// TIA Portal V17 export
// export: Created 2025-04-09T08:02:46.8788876Z, ExportSetting WithDefaults, DisplayName Totally Integrated Automation Portal, DisplayVersion V17 Update 8, DisplayName TIA Portal Openness, DisplayVersion V17 Update 8, DisplayName TIA Portal Version Control Interface, DisplayVersion V17, DisplayName SINAMICS Startdrive Advanced, DisplayVersion V17 SP2, DisplayName SINAMICS Startdrive G110M, G120, G120C, G120D, G120P, G115D, DisplayVersion V17 SP2, DisplayName SINAMICS Startdrive G130, G150, S120, S150, SINAMICS MV, S210, DisplayVersion V17 SP2, DisplayName STEP 7 Professional, DisplayVersion V17 Update 8, DisplayName SINUMERIK ONE STEP 7 Toolbox, DisplayVersion V17 Update 12, DisplayName SINUMERIK ONE PLC Basic Program Plus, DisplayVersion V17 Update 12, DisplayName SINUMERIK 840D sl STEP 7 Toolbox, DisplayVersion V17 Update 12, DisplayName STEP 7 Safety, DisplayVersion V17 Update 6, DisplayName WinCC Advanced, DisplayVersion V17 Update 8
FUNCTION_BLOCK "FB1701_KELLER_ASPIRATION_CONTROL"   // FB1701, LAD
{ S7_Optimized_Access := 'TRUE' }
VERSION : 0.1
// stored: AutoNumber false, IsIECCheckEnabled false, IsRetainMemResEnabled false, MemoryReserve 100, SetENOAutomatically false, UDAEnableTagReadback false
   VAR_INPUT
      IN_PRODUCTION { ExternalAccessible := 'False'; ExternalVisible := 'False'; ExternalWritable := 'False'} : Bool;   // EXTRACTION IN PRODUCTION
      NOT_FAULT { ExternalAccessible := 'False'; ExternalVisible := 'False'; ExternalWritable := 'False'} : Bool;   // EXTRACTION OK
      REQ_FILTER_CLEAN { ExternalAccessible := 'False'; ExternalVisible := 'False'; ExternalWritable := 'False'} : Bool;   // REQUEST FILTER CLEAN
      HMI_REQ_LINE { ExternalAccessible := 'False'; ExternalVisible := 'False'; ExternalWritable := 'False'} : Bool;   // HMI REQUEST LINE
      MACHINE_ALARM : Bool;
   END_VAR
   VAR_OUTPUT
      SWITCH_ON { ExternalAccessible := 'False'; ExternalVisible := 'False'; ExternalWritable := 'False'} : Bool;   // EXTRACTION SWITCH ON
      MACHINE_OK { ExternalAccessible := 'False'; ExternalVisible := 'False'; ExternalWritable := 'False'} : Bool;   // MACHINE OK
      ALLOW_CLEANING { ExternalAccessible := 'False'; ExternalVisible := 'False'; ExternalWritable := 'False'} : Bool;   // EXTRACTION ALLOW CLEANING
      HMI_POWER_UP_COND_OFF : Bool;   // HMI POWER UP CONDITIONS OFF
      HMI_POWER_UP_COND_ON : Bool;   // HMI POWER UP CONDITIONS ON
      HMI_POWER_UP_EXECU_LEFT : Bool;   // HMI POWER UP EXECUTABLE LEFT
      HMI_POWER_UP_EXECU_RIGHT : Bool;   // HMI POWER UP EXECUTABLE RIGHT
   END_VAR
   VAR DB_SPECIFIC
      SWITCH_ON_GENERAL_CONDITIONS : Bool;   // SWITCH ON GENERAL CONDITIONS
      SWITCH_ON_INITIAL_CONDITIONS : Bool;   // SWITCH ON INITIAL CONDITIONS
      SWITCH_ON_MANUAL_REQUEST : Bool;   // SWITCH ON MANUAL REQUEST
      SWITCH_ON_AUTO_REQUEST : Bool;   // SWITCH ON AUTO REQUEST
      SWITCH_ON_GLOBAL_REQUEST : Bool;   // SWITCH ON GLOBAL REQUEST
      SWITCH_ON_COMMAND : Bool;   // SWITCH ON COMMAND
      SWITCH_ON_1 : Bool;   // SWITCH ON
      IN_SERVICE : Bool;   // IN SERVICE
      SWITCH_OFF_GENERAL_CONDITIONS : Bool;   // SWITCH OFF GENERAL CONDITIONS
      SWITCH_OFF_INITIAL_CONDITIONS : Bool;   // SWITCH OFF INITIAL CONDITIONS
      SWITCH_OFF_MANUAL_REQUEST : Bool;   // SWITCH OFF MANUAL REQUEST
      SWITCH_OFF_AUTO_REQUEST : Bool;   // SWITCH OFF AUTO REQUEST
      SWITCH_OFF_GLOBAL_REQUEST : Bool;   // SWITCH OFF GLOBAL REQUEST
      SWITCH_OFF_COMMAND : Bool;   // SWITCH OFF COMMAND
      SWITCH_OFF : Bool;   // SWITCH OFF
      OUT_OF_SERVICE : Bool;   // OUT OF SERVICE
      RUNOUT_REQ_CLEAN_FILTER : Bool;   // RUNOUT REQUEST BY ASPIRATION SYSTEM TO CLEAN FILTERS
      MANUAL_REQUEST_HELP : Bool;   // MANUAL REQUEST HELP
      SWITCH_ON_GENERAL_CONDITION_HELP : Bool;   // SWITCH ON GENERAL CONDITION HELP
      SWITCH_ON_INITIAL_CONDITION_HELP : Bool;   // SWITCH ON INITIAL CONDITION HELP
      SWITCH_OFF_GENERAL_CONDITION_HELP : Bool;   // SWITCH OFF GENERAL CONDITION HELP
      SWITCH_OFF_INITIAL_CONDITION_HELP : Bool;   // SWITCH OFF INITIAL CONDITION HELP
      EXTRACTION_ALARM : Bool;   // EXTRACTION IN FAULT STATE
      ANY_ACTIVE_ALARM : Bool;   // ANY ACTIVE ALARM
      IS_ALARMS : Bool;   // IMMEDIATE STOP ALARMS
      SEOC_ALARMS : Bool;   // STOP END OF CYCLE ALARMS
      WARNINGS : Bool;   // WARNINGS
      WARNINGS_GONE : Bool;   // WARNINGS GONE
   END_VAR
   VAR_TEMP
      DB_NUMBER : DInt;   // DB NUMBER FOR ALARM DECODING
   END_VAR
   VAR_TEMP   // added for the SCL form of the ladder/FBD networks
      _w1 : Bool;
   END_VAR
BEGIN

NETWORK
TITLE = READ INSTANCE DB
      L     DINO;
      +     10#800000;
      T     #DB_NUMBER;


REGION Network 2: SWITCH GENERAL CONDITIONS
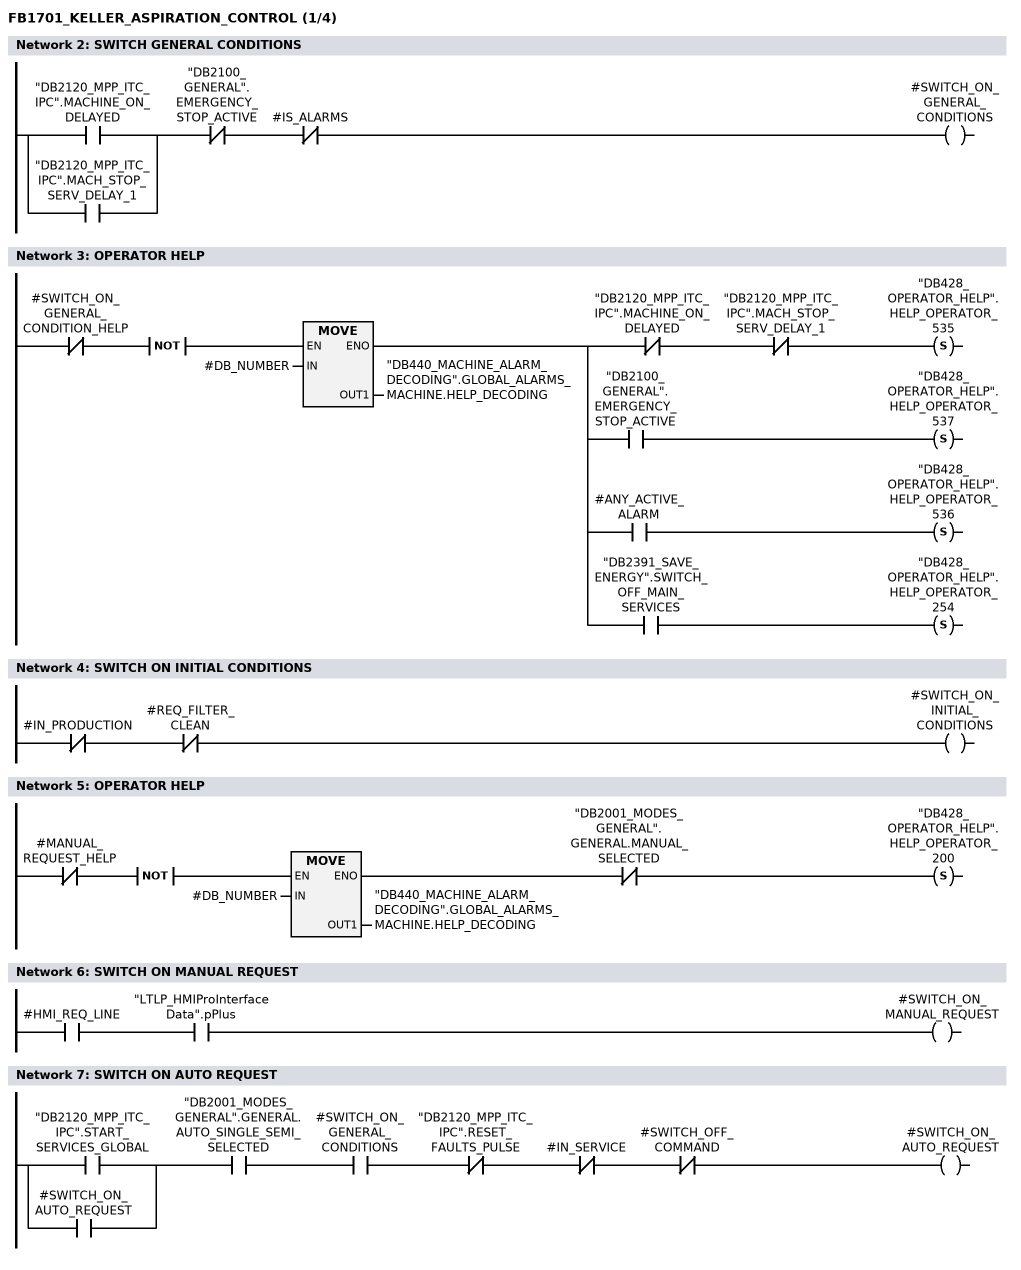
   RUNG wire#powerrail
      Contact( "DB2120_MPP_ITC_IPC".MACHINE_ON_DELAYED )
      wire#w1
      I_Contact( "DB2100_GENERAL".EMERGENCY_STOP_ACTIVE )
      I_Contact( #IS_ALARMS )
      Coil( #SWITCH_ON_GENERAL_CONDITIONS )
   END_RUNG
   RUNG wire#powerrail
      Contact( "DB2120_MPP_ITC_IPC".MACH_STOP_SERV_DELAY_1 )
   END_RUNG wire#w1
   // the same network as SCL:
   #SWITCH_ON_GENERAL_CONDITIONS := ("DB2120_MPP_ITC_IPC".MACHINE_ON_DELAYED OR "DB2120_MPP_ITC_IPC".MACH_STOP_SERV_DELAY_1) AND NOT "DB2100_GENERAL".EMERGENCY_STOP_ACTIVE AND NOT #IS_ALARMS;
END_REGION

REGION Network 3: OPERATOR HELP
   RUNG wire#powerrail
      I_Contact( #SWITCH_ON_GENERAL_CONDITION_HELP )
      Not()
      { S7_GenerateENO := "TRUE" } Move(in := #DB_NUMBER, out1 => "DB440_MACHINE_ALARM_DECODING".GLOBAL_ALARMS_MACHINE.HELP_DECODING)
      wire#w1
      I_Contact( "DB2120_MPP_ITC_IPC".MACHINE_ON_DELAYED )
      I_Contact( "DB2120_MPP_ITC_IPC".MACH_STOP_SERV_DELAY_1 )
      S_Coil( "DB428_OPERATOR_HELP".HELP_OPERATOR_535 )
   END_RUNG
   RUNG wire#w1
      Contact( "DB2100_GENERAL".EMERGENCY_STOP_ACTIVE )
      S_Coil( "DB428_OPERATOR_HELP".HELP_OPERATOR_537 )
   END_RUNG
   RUNG wire#w1
      Contact( #ANY_ACTIVE_ALARM )
      S_Coil( "DB428_OPERATOR_HELP".HELP_OPERATOR_536 )
   END_RUNG
   RUNG wire#w1
      Contact( "DB2391_SAVE_ENERGY".SWITCH_OFF_MAIN_SERVICES )
      S_Coil( "DB428_OPERATOR_HELP".HELP_OPERATOR_254 )
   END_RUNG
   // the same network as SCL:
   // ENO of a box is taken as its EN; it also drops when the box reports an error
   #_w1 := NOT (NOT #SWITCH_ON_GENERAL_CONDITION_HELP);
   IF #_w1 THEN "DB440_MACHINE_ALARM_DECODING".GLOBAL_ALARMS_MACHINE.HELP_DECODING := #DB_NUMBER; END_IF;
   IF #_w1 AND NOT "DB2120_MPP_ITC_IPC".MACHINE_ON_DELAYED AND NOT "DB2120_MPP_ITC_IPC".MACH_STOP_SERV_DELAY_1 THEN
       "DB428_OPERATOR_HELP".HELP_OPERATOR_535 := TRUE;
   END_IF;
   IF #_w1 AND "DB2100_GENERAL".EMERGENCY_STOP_ACTIVE THEN
       "DB428_OPERATOR_HELP".HELP_OPERATOR_537 := TRUE;
   END_IF;
   IF #_w1 AND #ANY_ACTIVE_ALARM THEN "DB428_OPERATOR_HELP".HELP_OPERATOR_536 := TRUE; END_IF;
   IF #_w1 AND "DB2391_SAVE_ENERGY".SWITCH_OFF_MAIN_SERVICES THEN
       "DB428_OPERATOR_HELP".HELP_OPERATOR_254 := TRUE;
   END_IF;
END_REGION

REGION Network 4: SWITCH ON INITIAL CONDITIONS
   RUNG wire#powerrail
      I_Contact( #IN_PRODUCTION )
      I_Contact( #REQ_FILTER_CLEAN )
      Coil( #SWITCH_ON_INITIAL_CONDITIONS )
   END_RUNG
   // the same network as SCL:
   #SWITCH_ON_INITIAL_CONDITIONS := NOT #IN_PRODUCTION AND NOT #REQ_FILTER_CLEAN;
END_REGION

REGION Network 5: OPERATOR HELP
   RUNG wire#powerrail
      I_Contact( #MANUAL_REQUEST_HELP )
      Not()
      { S7_GenerateENO := "TRUE" } Move(in := #DB_NUMBER, out1 => "DB440_MACHINE_ALARM_DECODING".GLOBAL_ALARMS_MACHINE.HELP_DECODING)
      I_Contact( "DB2001_MODES_GENERAL".GENERAL.MANUAL_SELECTED )
      S_Coil( "DB428_OPERATOR_HELP".HELP_OPERATOR_200 )
   END_RUNG
   // the same network as SCL:
   // ENO of a box is taken as its EN; it also drops when the box reports an error
   #_w1 := NOT (NOT #MANUAL_REQUEST_HELP);
   IF #_w1 THEN "DB440_MACHINE_ALARM_DECODING".GLOBAL_ALARMS_MACHINE.HELP_DECODING := #DB_NUMBER; END_IF;
   IF #_w1 AND NOT "DB2001_MODES_GENERAL".GENERAL.MANUAL_SELECTED THEN
       "DB428_OPERATOR_HELP".HELP_OPERATOR_200 := TRUE;
   END_IF;
END_REGION

REGION Network 6: SWITCH ON MANUAL REQUEST
   RUNG wire#powerrail
      Contact( #HMI_REQ_LINE )
      Contact( "LTLP_HMIProInterfaceData".pPlus )
      Coil( #SWITCH_ON_MANUAL_REQUEST )
   END_RUNG
   // the same network as SCL:
   #SWITCH_ON_MANUAL_REQUEST := #HMI_REQ_LINE AND "LTLP_HMIProInterfaceData".pPlus;
END_REGION

REGION Network 7: SWITCH ON AUTO REQUEST
   RUNG wire#powerrail
      Contact( "DB2120_MPP_ITC_IPC".START_SERVICES_GLOBAL )
      wire#w1
      Contact( "DB2001_MODES_GENERAL".GENERAL.AUTO_SINGLE_SEMI_SELECTED )
      Contact( #SWITCH_ON_GENERAL_CONDITIONS )
      I_Contact( "DB2120_MPP_ITC_IPC".RESET_FAULTS_PULSE )
      I_Contact( #IN_SERVICE )
      I_Contact( #SWITCH_OFF_COMMAND )
      Coil( #SWITCH_ON_AUTO_REQUEST )
   END_RUNG
   RUNG wire#powerrail
      Contact( #SWITCH_ON_AUTO_REQUEST )
   END_RUNG wire#w1
   // the same network as SCL:
   #SWITCH_ON_AUTO_REQUEST := ("DB2120_MPP_ITC_IPC".START_SERVICES_GLOBAL OR #SWITCH_ON_AUTO_REQUEST) AND "DB2001_MODES_GENERAL".GENERAL.AUTO_SINGLE_SEMI_SELECTED AND #SWITCH_ON_GENERAL_CONDITIONS AND NOT "DB2120_MPP_ITC_IPC".RESET_FAULTS_PULSE AND NOT #IN_SERVICE AND NOT #SWITCH_OFF_COMMAND;
END_REGION

REGION Network 8: SWITCH ON GLOBAL REQUEST
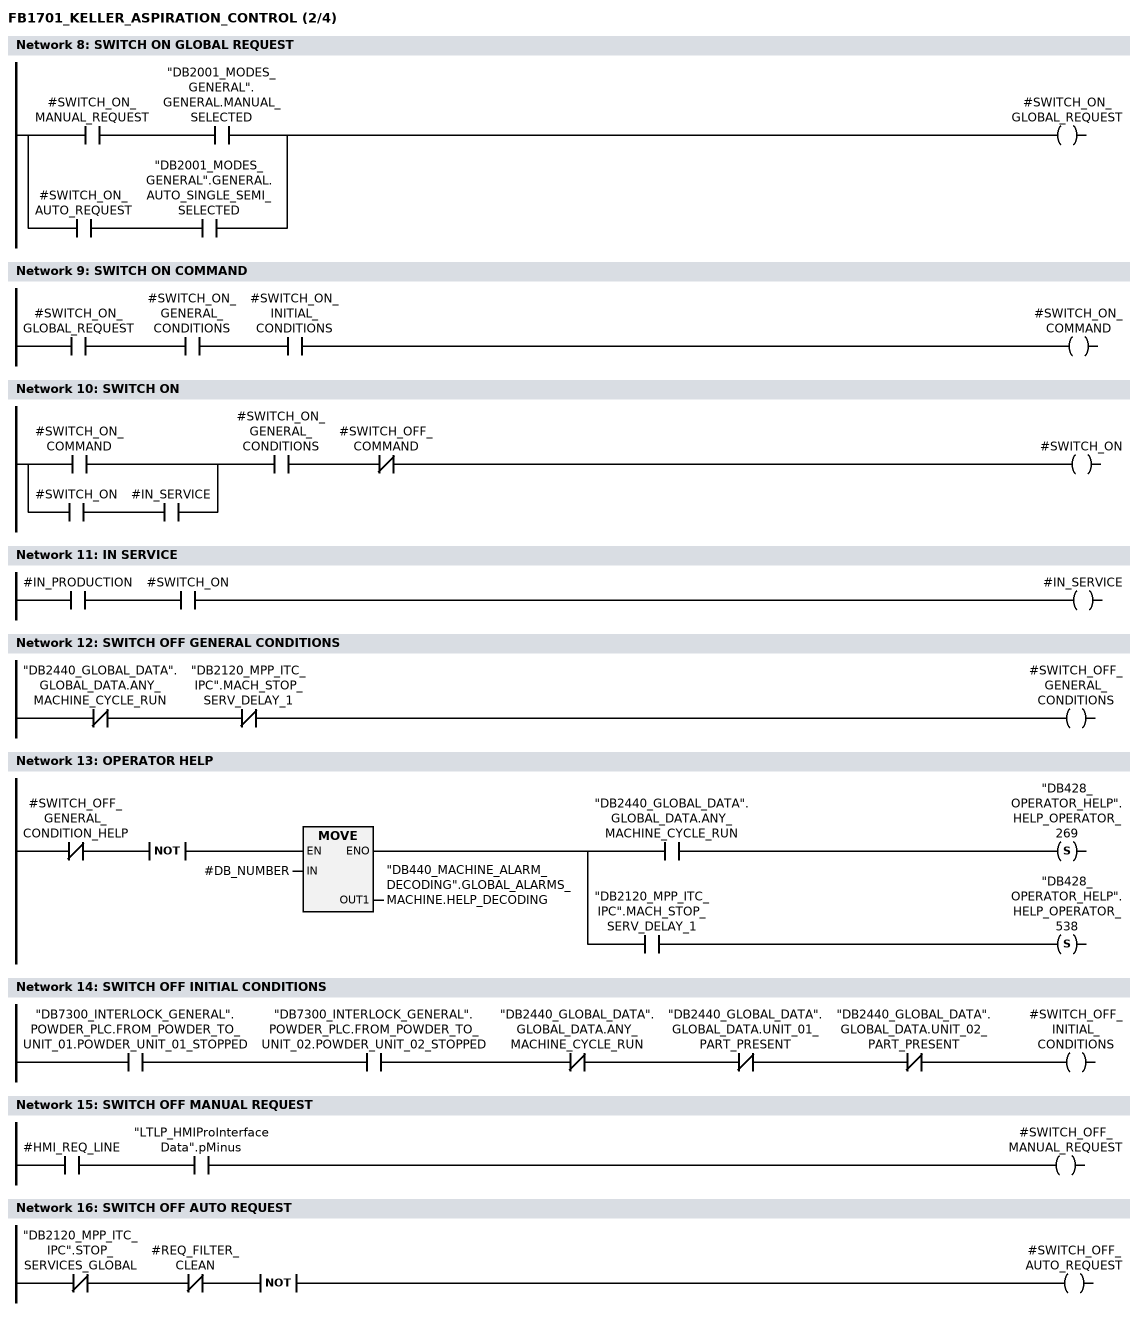
   RUNG wire#powerrail
      Contact( #SWITCH_ON_MANUAL_REQUEST )
      Contact( "DB2001_MODES_GENERAL".GENERAL.MANUAL_SELECTED )
      wire#w1
      Coil( #SWITCH_ON_GLOBAL_REQUEST )
   END_RUNG
   RUNG wire#powerrail
      Contact( #SWITCH_ON_AUTO_REQUEST )
      Contact( "DB2001_MODES_GENERAL".GENERAL.AUTO_SINGLE_SEMI_SELECTED )
   END_RUNG wire#w1
   // the same network as SCL:
   #SWITCH_ON_GLOBAL_REQUEST := (#SWITCH_ON_MANUAL_REQUEST AND "DB2001_MODES_GENERAL".GENERAL.MANUAL_SELECTED) OR (#SWITCH_ON_AUTO_REQUEST AND "DB2001_MODES_GENERAL".GENERAL.AUTO_SINGLE_SEMI_SELECTED);
END_REGION

REGION Network 9: SWITCH ON COMMAND
   RUNG wire#powerrail
      Contact( #SWITCH_ON_GLOBAL_REQUEST )
      Contact( #SWITCH_ON_GENERAL_CONDITIONS )
      Contact( #SWITCH_ON_INITIAL_CONDITIONS )
      Coil( #SWITCH_ON_COMMAND )
   END_RUNG
   // the same network as SCL:
   #SWITCH_ON_COMMAND := #SWITCH_ON_GLOBAL_REQUEST AND #SWITCH_ON_GENERAL_CONDITIONS AND #SWITCH_ON_INITIAL_CONDITIONS;
END_REGION

REGION Network 10: SWITCH ON
   RUNG wire#powerrail
      Contact( #SWITCH_ON_COMMAND )
      wire#w1
      Contact( #SWITCH_ON_GENERAL_CONDITIONS )
      I_Contact( #SWITCH_OFF_COMMAND )
      Coil( #SWITCH_ON )
   END_RUNG
   RUNG wire#powerrail
      Contact( #SWITCH_ON )
      Contact( #IN_SERVICE )
   END_RUNG wire#w1
   // the same network as SCL:
   #SWITCH_ON := (#SWITCH_ON_COMMAND OR (#SWITCH_ON AND #IN_SERVICE)) AND #SWITCH_ON_GENERAL_CONDITIONS AND NOT #SWITCH_OFF_COMMAND;
END_REGION

REGION Network 11: IN SERVICE
   RUNG wire#powerrail
      Contact( #IN_PRODUCTION )
      Contact( #SWITCH_ON )
      Coil( #IN_SERVICE )
   END_RUNG
   // the same network as SCL:
   #IN_SERVICE := #IN_PRODUCTION AND #SWITCH_ON;
END_REGION

REGION Network 12: SWITCH OFF GENERAL CONDITIONS
   RUNG wire#powerrail
      I_Contact( "DB2440_GLOBAL_DATA".GLOBAL_DATA.ANY_MACHINE_CYCLE_RUN )
      I_Contact( "DB2120_MPP_ITC_IPC".MACH_STOP_SERV_DELAY_1 )
      Coil( #SWITCH_OFF_GENERAL_CONDITIONS )
   END_RUNG
   // the same network as SCL:
   #SWITCH_OFF_GENERAL_CONDITIONS := NOT "DB2440_GLOBAL_DATA".GLOBAL_DATA.ANY_MACHINE_CYCLE_RUN AND NOT "DB2120_MPP_ITC_IPC".MACH_STOP_SERV_DELAY_1;
END_REGION

REGION Network 13: OPERATOR HELP
   RUNG wire#powerrail
      I_Contact( #SWITCH_OFF_GENERAL_CONDITION_HELP )
      Not()
      { S7_GenerateENO := "TRUE" } Move(in := #DB_NUMBER, out1 => "DB440_MACHINE_ALARM_DECODING".GLOBAL_ALARMS_MACHINE.HELP_DECODING)
      wire#w1
      Contact( "DB2440_GLOBAL_DATA".GLOBAL_DATA.ANY_MACHINE_CYCLE_RUN )
      S_Coil( "DB428_OPERATOR_HELP".HELP_OPERATOR_269 )
   END_RUNG
   RUNG wire#w1
      Contact( "DB2120_MPP_ITC_IPC".MACH_STOP_SERV_DELAY_1 )
      S_Coil( "DB428_OPERATOR_HELP".HELP_OPERATOR_538 )
   END_RUNG
   // the same network as SCL:
   // ENO of a box is taken as its EN; it also drops when the box reports an error
   #_w1 := NOT (NOT #SWITCH_OFF_GENERAL_CONDITION_HELP);
   IF #_w1 THEN "DB440_MACHINE_ALARM_DECODING".GLOBAL_ALARMS_MACHINE.HELP_DECODING := #DB_NUMBER; END_IF;
   IF #_w1 AND "DB2440_GLOBAL_DATA".GLOBAL_DATA.ANY_MACHINE_CYCLE_RUN THEN
       "DB428_OPERATOR_HELP".HELP_OPERATOR_269 := TRUE;
   END_IF;
   IF #_w1 AND "DB2120_MPP_ITC_IPC".MACH_STOP_SERV_DELAY_1 THEN
       "DB428_OPERATOR_HELP".HELP_OPERATOR_538 := TRUE;
   END_IF;
END_REGION

REGION Network 14: SWITCH OFF INITIAL CONDITIONS
   RUNG wire#powerrail
      Contact( "DB7300_INTERLOCK_GENERAL".POWDER_PLC.FROM_POWDER_TO_UNIT_01.POWDER_UNIT_01_STOPPED )
      Contact( "DB7300_INTERLOCK_GENERAL".POWDER_PLC.FROM_POWDER_TO_UNIT_02.POWDER_UNIT_02_STOPPED )
      I_Contact( "DB2440_GLOBAL_DATA".GLOBAL_DATA.ANY_MACHINE_CYCLE_RUN )
      I_Contact( "DB2440_GLOBAL_DATA".GLOBAL_DATA.UNIT_01_PART_PRESENT )
      I_Contact( "DB2440_GLOBAL_DATA".GLOBAL_DATA.UNIT_02_PART_PRESENT )
      Coil( #SWITCH_OFF_INITIAL_CONDITIONS )
   END_RUNG
   // the same network as SCL:
   #SWITCH_OFF_INITIAL_CONDITIONS := "DB7300_INTERLOCK_GENERAL".POWDER_PLC.FROM_POWDER_TO_UNIT_01.POWDER_UNIT_01_STOPPED AND "DB7300_INTERLOCK_GENERAL".POWDER_PLC.FROM_POWDER_TO_UNIT_02.POWDER_UNIT_02_STOPPED AND NOT "DB2440_GLOBAL_DATA".GLOBAL_DATA.ANY_MACHINE_CYCLE_RUN AND NOT "DB2440_GLOBAL_DATA".GLOBAL_DATA.UNIT_01_PART_PRESENT AND NOT "DB2440_GLOBAL_DATA".GLOBAL_DATA.UNIT_02_PART_PRESENT;
END_REGION

REGION Network 15: SWITCH OFF MANUAL REQUEST
   RUNG wire#powerrail
      Contact( #HMI_REQ_LINE )
      Contact( "LTLP_HMIProInterfaceData".pMinus )
      Coil( #SWITCH_OFF_MANUAL_REQUEST )
   END_RUNG
   // the same network as SCL:
   #SWITCH_OFF_MANUAL_REQUEST := #HMI_REQ_LINE AND "LTLP_HMIProInterfaceData".pMinus;
END_REGION

REGION Network 16: SWITCH OFF AUTO REQUEST
   RUNG wire#powerrail
      I_Contact( "DB2120_MPP_ITC_IPC".STOP_SERVICES_GLOBAL )
      I_Contact( #REQ_FILTER_CLEAN )
      Not()
      Coil( #SWITCH_OFF_AUTO_REQUEST )
   END_RUNG
   // the same network as SCL:
   #SWITCH_OFF_AUTO_REQUEST := NOT (NOT "DB2120_MPP_ITC_IPC".STOP_SERVICES_GLOBAL AND NOT #REQ_FILTER_CLEAN);
END_REGION

REGION Network 17: SWITCH OFF GLOBAL REQUEST
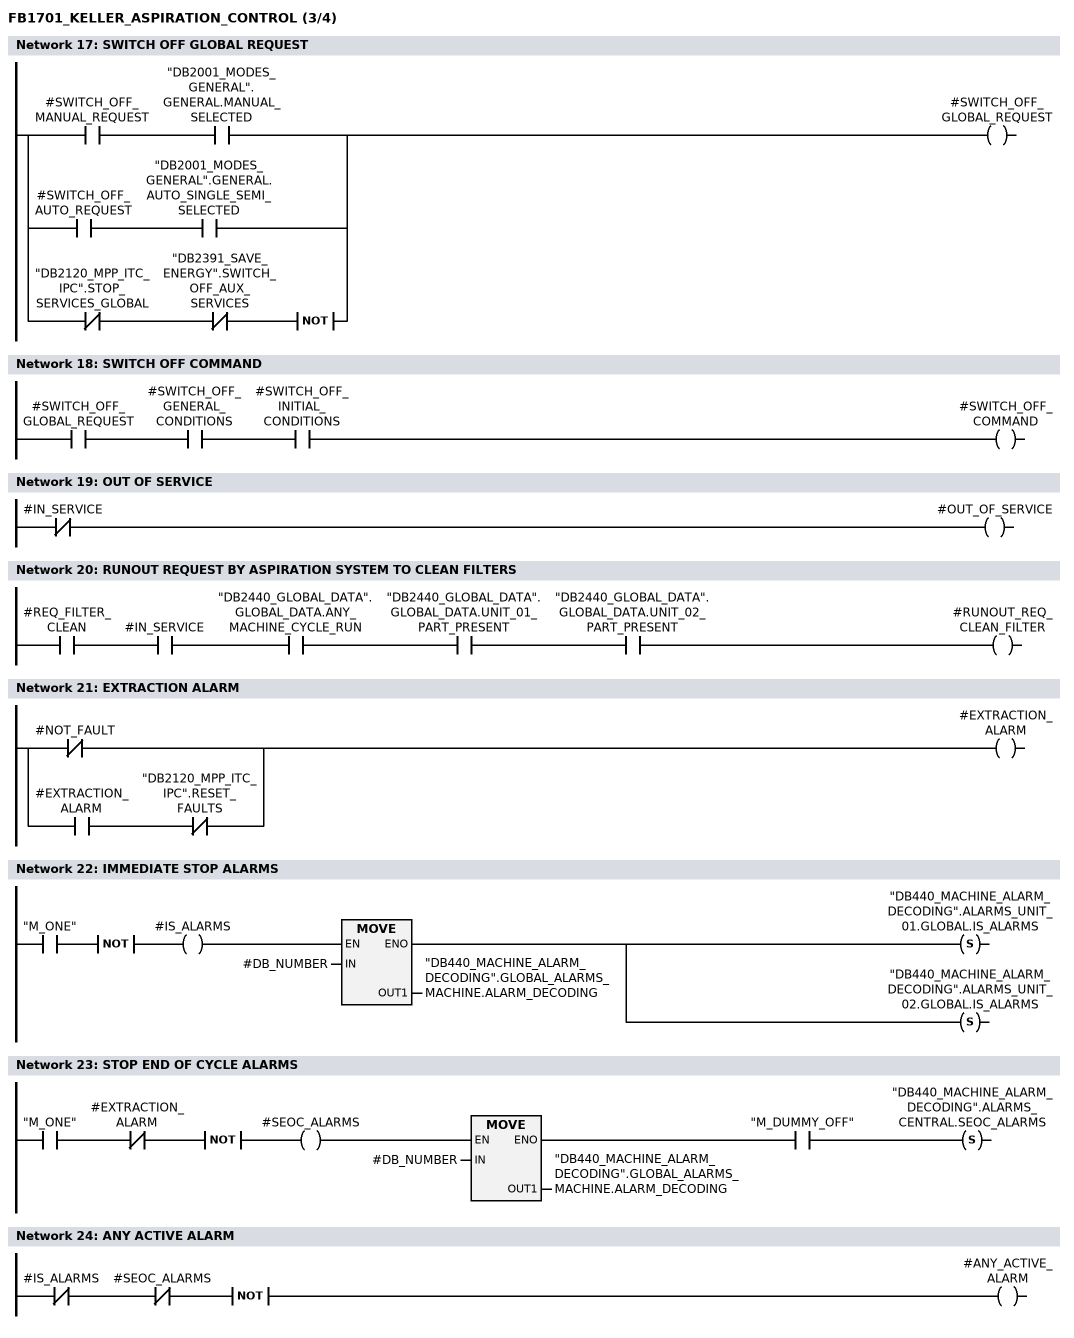
   RUNG wire#powerrail
      Contact( #SWITCH_OFF_MANUAL_REQUEST )
      Contact( "DB2001_MODES_GENERAL".GENERAL.MANUAL_SELECTED )
      wire#w1
      Coil( #SWITCH_OFF_GLOBAL_REQUEST )
   END_RUNG
   RUNG wire#powerrail
      Contact( #SWITCH_OFF_AUTO_REQUEST )
      Contact( "DB2001_MODES_GENERAL".GENERAL.AUTO_SINGLE_SEMI_SELECTED )
   END_RUNG wire#w1
   RUNG wire#powerrail
      I_Contact( "DB2120_MPP_ITC_IPC".STOP_SERVICES_GLOBAL )
      I_Contact( "DB2391_SAVE_ENERGY".SWITCH_OFF_AUX_SERVICES )
      Not()
   END_RUNG wire#w1
   // the same network as SCL:
   #SWITCH_OFF_GLOBAL_REQUEST := (#SWITCH_OFF_MANUAL_REQUEST AND "DB2001_MODES_GENERAL".GENERAL.MANUAL_SELECTED) OR (#SWITCH_OFF_AUTO_REQUEST AND "DB2001_MODES_GENERAL".GENERAL.AUTO_SINGLE_SEMI_SELECTED) OR NOT (NOT "DB2120_MPP_ITC_IPC".STOP_SERVICES_GLOBAL AND NOT "DB2391_SAVE_ENERGY".SWITCH_OFF_AUX_SERVICES);
END_REGION

REGION Network 18: SWITCH OFF COMMAND
   RUNG wire#powerrail
      Contact( #SWITCH_OFF_GLOBAL_REQUEST )
      Contact( #SWITCH_OFF_GENERAL_CONDITIONS )
      Contact( #SWITCH_OFF_INITIAL_CONDITIONS )
      Coil( #SWITCH_OFF_COMMAND )
   END_RUNG
   // the same network as SCL:
   #SWITCH_OFF_COMMAND := #SWITCH_OFF_GLOBAL_REQUEST AND #SWITCH_OFF_GENERAL_CONDITIONS AND #SWITCH_OFF_INITIAL_CONDITIONS;
END_REGION

REGION Network 19: OUT OF SERVICE
   RUNG wire#powerrail
      I_Contact( #IN_SERVICE )
      Coil( #OUT_OF_SERVICE )
   END_RUNG
   // the same network as SCL:
   #OUT_OF_SERVICE := NOT #IN_SERVICE;
END_REGION

REGION Network 20: RUNOUT REQUEST BY ASPIRATION SYSTEM TO CLEAN FILTERS
   RUNG wire#powerrail
      Contact( #REQ_FILTER_CLEAN )
      Contact( #IN_SERVICE )
      Contact( "DB2440_GLOBAL_DATA".GLOBAL_DATA.ANY_MACHINE_CYCLE_RUN )
      Contact( "DB2440_GLOBAL_DATA".GLOBAL_DATA.UNIT_01_PART_PRESENT )
      Contact( "DB2440_GLOBAL_DATA".GLOBAL_DATA.UNIT_02_PART_PRESENT )
      Coil( #RUNOUT_REQ_CLEAN_FILTER )
   END_RUNG
   // the same network as SCL:
   #RUNOUT_REQ_CLEAN_FILTER := #REQ_FILTER_CLEAN AND #IN_SERVICE AND "DB2440_GLOBAL_DATA".GLOBAL_DATA.ANY_MACHINE_CYCLE_RUN AND "DB2440_GLOBAL_DATA".GLOBAL_DATA.UNIT_01_PART_PRESENT AND "DB2440_GLOBAL_DATA".GLOBAL_DATA.UNIT_02_PART_PRESENT;
END_REGION

REGION Network 21: EXTRACTION ALARM
   RUNG wire#powerrail
      I_Contact( #NOT_FAULT )
      wire#w1
      Coil( #EXTRACTION_ALARM )
   END_RUNG
   RUNG wire#powerrail
      Contact( #EXTRACTION_ALARM )
      I_Contact( "DB2120_MPP_ITC_IPC".RESET_FAULTS )
   END_RUNG wire#w1
   // the same network as SCL:
   #EXTRACTION_ALARM := NOT #NOT_FAULT OR (#EXTRACTION_ALARM AND NOT "DB2120_MPP_ITC_IPC".RESET_FAULTS);
END_REGION

REGION Network 22: IMMEDIATE STOP ALARMS
   RUNG wire#powerrail
      Contact( "M_ONE" )
      Not()
      Coil( #IS_ALARMS )
      Move(in := #DB_NUMBER, out1 => "DB440_MACHINE_ALARM_DECODING".GLOBAL_ALARMS_MACHINE.ALARM_DECODING)
      wire#w1
      S_Coil( "DB440_MACHINE_ALARM_DECODING".ALARMS_UNIT_01.GLOBAL.IS_ALARMS )
   END_RUNG
   RUNG wire#w1
      S_Coil( "DB440_MACHINE_ALARM_DECODING".ALARMS_UNIT_02.GLOBAL.IS_ALARMS )
   END_RUNG
   // the same network as SCL:
   #IS_ALARMS := NOT "M_ONE";
   IF NOT "M_ONE" THEN
       "DB440_MACHINE_ALARM_DECODING".GLOBAL_ALARMS_MACHINE.ALARM_DECODING := #DB_NUMBER;
       "DB440_MACHINE_ALARM_DECODING".ALARMS_UNIT_01.GLOBAL.IS_ALARMS := TRUE;
       "DB440_MACHINE_ALARM_DECODING".ALARMS_UNIT_02.GLOBAL.IS_ALARMS := TRUE;
   END_IF;
END_REGION

REGION Network 23: STOP END OF CYCLE ALARMS
   RUNG wire#powerrail
      Contact( "M_ONE" )
      I_Contact( #EXTRACTION_ALARM )
      Not()
      Coil( #SEOC_ALARMS )
      Move(in := #DB_NUMBER, out1 => "DB440_MACHINE_ALARM_DECODING".GLOBAL_ALARMS_MACHINE.ALARM_DECODING)
      Contact( "M_DUMMY_OFF" )
      S_Coil( "DB440_MACHINE_ALARM_DECODING".ALARMS_CENTRAL.SEOC_ALARMS )
   END_RUNG
   // the same network as SCL:
   #SEOC_ALARMS := NOT ("M_ONE" AND NOT #EXTRACTION_ALARM);
   IF #SEOC_ALARMS THEN
       "DB440_MACHINE_ALARM_DECODING".GLOBAL_ALARMS_MACHINE.ALARM_DECODING := #DB_NUMBER;
   END_IF;
   IF #SEOC_ALARMS AND "M_DUMMY_OFF" THEN
       "DB440_MACHINE_ALARM_DECODING".ALARMS_CENTRAL.SEOC_ALARMS := TRUE;
   END_IF;
END_REGION

REGION Network 24: ANY ACTIVE ALARM
   RUNG wire#powerrail
      I_Contact( #IS_ALARMS )
      I_Contact( #SEOC_ALARMS )
      Not()
      Coil( #ANY_ACTIVE_ALARM )
   END_RUNG
   // the same network as SCL:
   #ANY_ACTIVE_ALARM := NOT (NOT #IS_ALARMS AND NOT #SEOC_ALARMS);
END_REGION

REGION Network 25: MANUAL REQUEST HELP
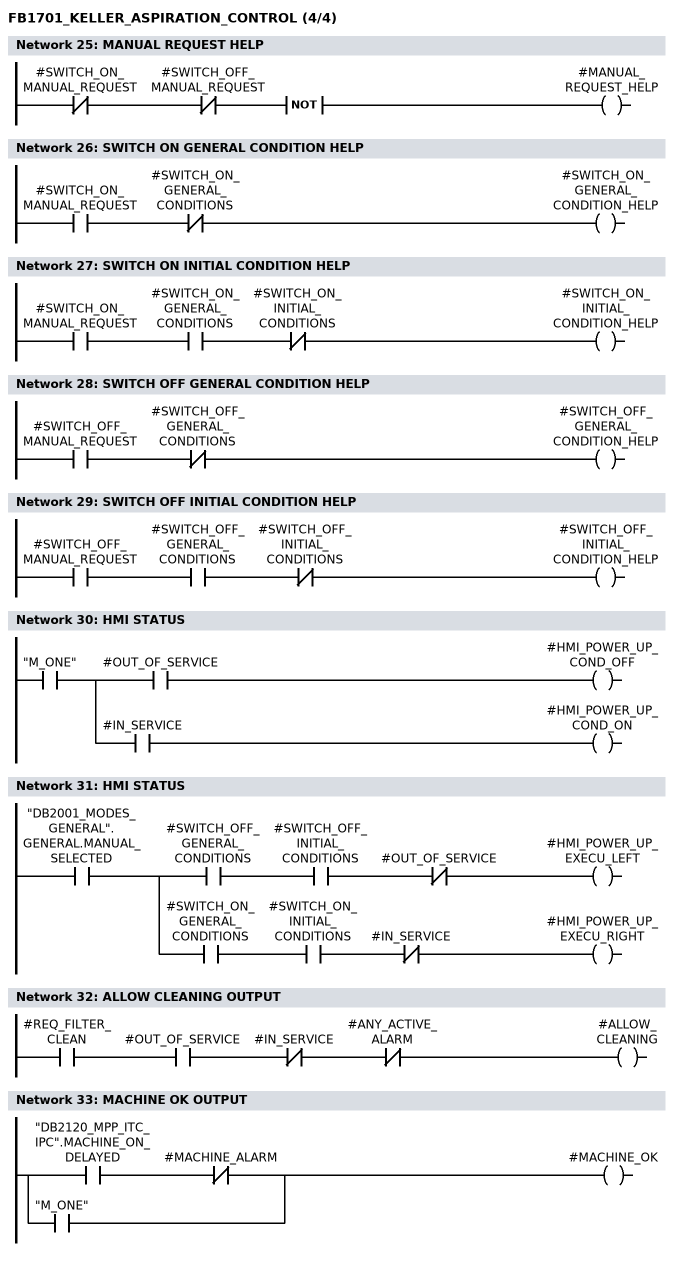
   RUNG wire#powerrail
      I_Contact( #SWITCH_ON_MANUAL_REQUEST )
      I_Contact( #SWITCH_OFF_MANUAL_REQUEST )
      Not()
      Coil( #MANUAL_REQUEST_HELP )
   END_RUNG
   // the same network as SCL:
   #MANUAL_REQUEST_HELP := NOT (NOT #SWITCH_ON_MANUAL_REQUEST AND NOT #SWITCH_OFF_MANUAL_REQUEST);
END_REGION

REGION Network 26: SWITCH ON GENERAL CONDITION HELP
   RUNG wire#powerrail
      Contact( #SWITCH_ON_MANUAL_REQUEST )
      I_Contact( #SWITCH_ON_GENERAL_CONDITIONS )
      Coil( #SWITCH_ON_GENERAL_CONDITION_HELP )
   END_RUNG
   // the same network as SCL:
   #SWITCH_ON_GENERAL_CONDITION_HELP := #SWITCH_ON_MANUAL_REQUEST AND NOT #SWITCH_ON_GENERAL_CONDITIONS;
END_REGION

REGION Network 27: SWITCH ON INITIAL CONDITION HELP
   RUNG wire#powerrail
      Contact( #SWITCH_ON_MANUAL_REQUEST )
      Contact( #SWITCH_ON_GENERAL_CONDITIONS )
      I_Contact( #SWITCH_ON_INITIAL_CONDITIONS )
      Coil( #SWITCH_ON_INITIAL_CONDITION_HELP )
   END_RUNG
   // the same network as SCL:
   #SWITCH_ON_INITIAL_CONDITION_HELP := #SWITCH_ON_MANUAL_REQUEST AND #SWITCH_ON_GENERAL_CONDITIONS AND NOT #SWITCH_ON_INITIAL_CONDITIONS;
END_REGION

REGION Network 28: SWITCH OFF GENERAL CONDITION HELP
   RUNG wire#powerrail
      Contact( #SWITCH_OFF_MANUAL_REQUEST )
      I_Contact( #SWITCH_OFF_GENERAL_CONDITIONS )
      Coil( #SWITCH_OFF_GENERAL_CONDITION_HELP )
   END_RUNG
   // the same network as SCL:
   #SWITCH_OFF_GENERAL_CONDITION_HELP := #SWITCH_OFF_MANUAL_REQUEST AND NOT #SWITCH_OFF_GENERAL_CONDITIONS;
END_REGION

REGION Network 29: SWITCH OFF INITIAL CONDITION HELP
   RUNG wire#powerrail
      Contact( #SWITCH_OFF_MANUAL_REQUEST )
      Contact( #SWITCH_OFF_GENERAL_CONDITIONS )
      I_Contact( #SWITCH_OFF_INITIAL_CONDITIONS )
      Coil( #SWITCH_OFF_INITIAL_CONDITION_HELP )
   END_RUNG
   // the same network as SCL:
   #SWITCH_OFF_INITIAL_CONDITION_HELP := #SWITCH_OFF_MANUAL_REQUEST AND #SWITCH_OFF_GENERAL_CONDITIONS AND NOT #SWITCH_OFF_INITIAL_CONDITIONS;
END_REGION

REGION Network 30: HMI STATUS
   RUNG wire#powerrail
      Contact( "M_ONE" )
      wire#w1
      Contact( #OUT_OF_SERVICE )
      Coil( #HMI_POWER_UP_COND_OFF )
   END_RUNG
   RUNG wire#w1
      Contact( #IN_SERVICE )
      Coil( #HMI_POWER_UP_COND_ON )
   END_RUNG
   // the same network as SCL:
   #HMI_POWER_UP_COND_OFF := "M_ONE" AND #OUT_OF_SERVICE;
   #HMI_POWER_UP_COND_ON := "M_ONE" AND #IN_SERVICE;
END_REGION

REGION Network 31: HMI STATUS
   RUNG wire#powerrail
      Contact( "DB2001_MODES_GENERAL".GENERAL.MANUAL_SELECTED )
      wire#w1
      Contact( #SWITCH_OFF_GENERAL_CONDITIONS )
      Contact( #SWITCH_OFF_INITIAL_CONDITIONS )
      I_Contact( #OUT_OF_SERVICE )
      Coil( #HMI_POWER_UP_EXECU_LEFT )
   END_RUNG
   RUNG wire#w1
      Contact( #SWITCH_ON_GENERAL_CONDITIONS )
      Contact( #SWITCH_ON_INITIAL_CONDITIONS )
      I_Contact( #IN_SERVICE )
      Coil( #HMI_POWER_UP_EXECU_RIGHT )
   END_RUNG
   // the same network as SCL:
   #HMI_POWER_UP_EXECU_LEFT := "DB2001_MODES_GENERAL".GENERAL.MANUAL_SELECTED AND #SWITCH_OFF_GENERAL_CONDITIONS AND #SWITCH_OFF_INITIAL_CONDITIONS AND NOT #OUT_OF_SERVICE;
   #HMI_POWER_UP_EXECU_RIGHT := "DB2001_MODES_GENERAL".GENERAL.MANUAL_SELECTED AND #SWITCH_ON_GENERAL_CONDITIONS AND #SWITCH_ON_INITIAL_CONDITIONS AND NOT #IN_SERVICE;
END_REGION

REGION Network 32: ALLOW CLEANING OUTPUT
   RUNG wire#powerrail
      Contact( #REQ_FILTER_CLEAN )
      Contact( #OUT_OF_SERVICE )
      I_Contact( #IN_SERVICE )
      I_Contact( #ANY_ACTIVE_ALARM )
      Coil( #ALLOW_CLEANING )
   END_RUNG
   // the same network as SCL:
   #ALLOW_CLEANING := #REQ_FILTER_CLEAN AND #OUT_OF_SERVICE AND NOT #IN_SERVICE AND NOT #ANY_ACTIVE_ALARM;
END_REGION

REGION Network 33: MACHINE OK OUTPUT
   RUNG wire#powerrail
      Contact( "DB2120_MPP_ITC_IPC".MACHINE_ON_DELAYED )
      I_Contact( #MACHINE_ALARM )
      wire#w1
      Coil( #MACHINE_OK )
   END_RUNG
   RUNG wire#powerrail
      Contact( "M_ONE" )
   END_RUNG wire#w1
   // the same network as SCL:
   #MACHINE_OK := ("DB2120_MPP_ITC_IPC".MACHINE_ON_DELAYED AND NOT #MACHINE_ALARM) OR "M_ONE";
END_REGION
END_FUNCTION_BLOCK
